REGION Network 65: UNIT 2 STATION 2 MISSING CALIBRATION IN FIXTURE 1 ALARM
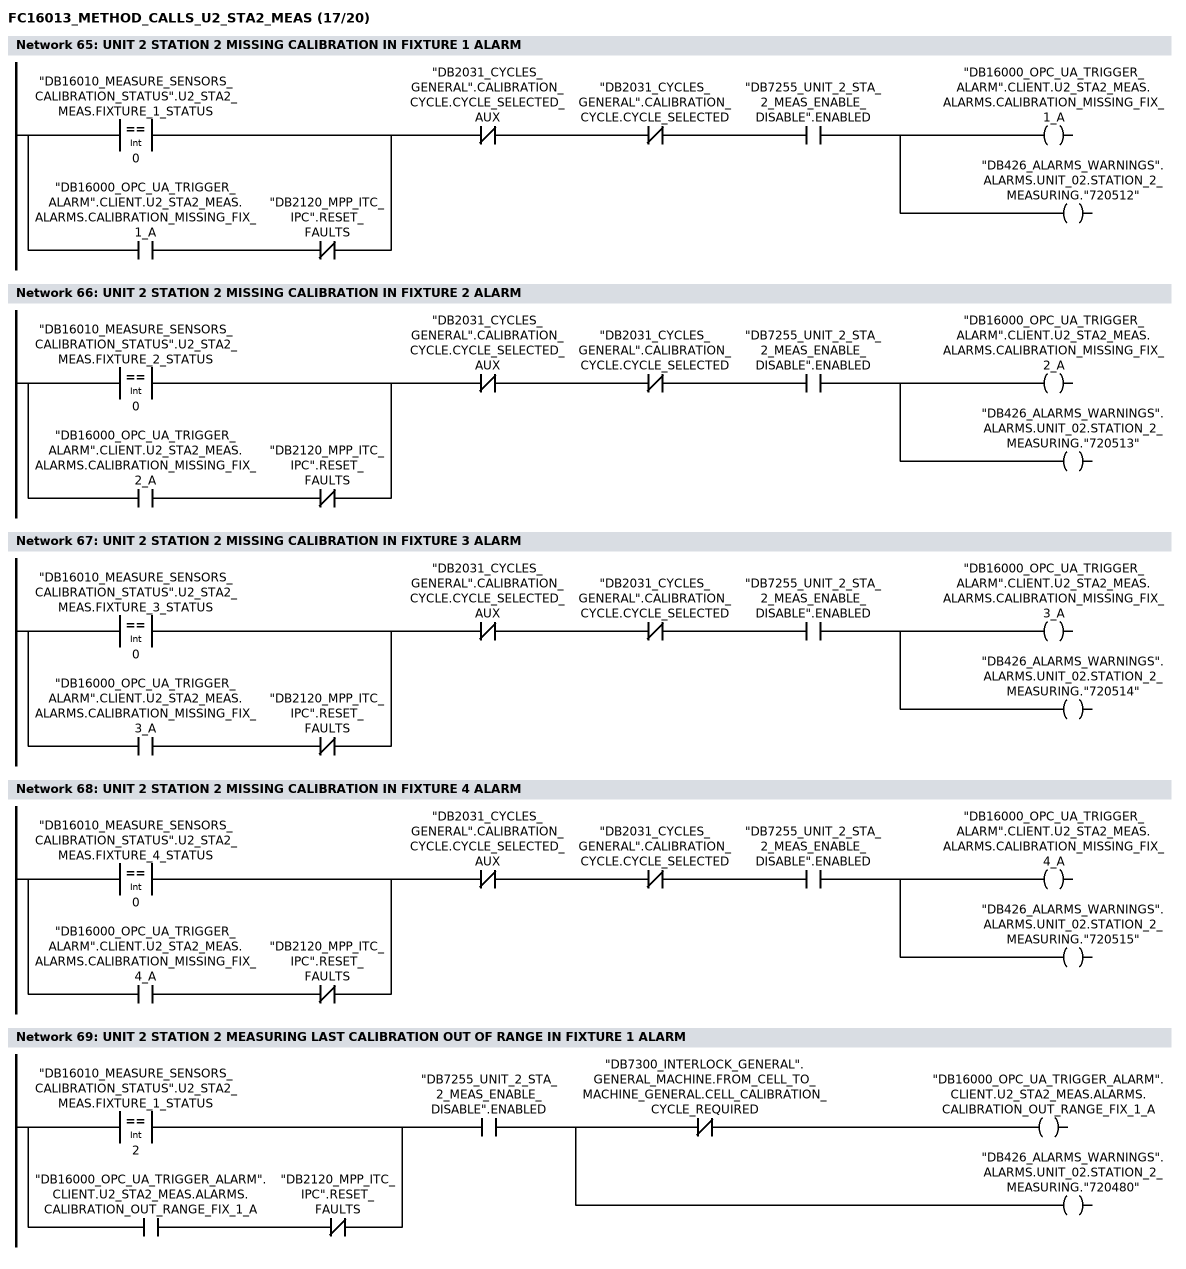
   RUNG wire#powerrail
      { S7_Templates := "SrcType := Int" } EQ_Contact(in1 := "DB16010_MEASURE_SENSORS_CALIBRATION_STATUS".U2_STA2_MEAS.FIXTURE_1_STATUS, in2 := 0)
      wire#w1
      I_Contact( "DB2031_CYCLES_GENERAL".CALIBRATION_CYCLE.CYCLE_SELECTED_AUX )
      I_Contact( "DB2031_CYCLES_GENERAL".CALIBRATION_CYCLE.CYCLE_SELECTED )
      Contact( "DB7255_UNIT_2_STA_2_MEAS_ENABLE_DISABLE".ENABLED )
      wire#w2
      Coil( "DB16000_OPC_UA_TRIGGER_ALARM".CLIENT.U2_STA2_MEAS.ALARMS.CALIBRATION_MISSING_FIX_1_A )
   END_RUNG
   RUNG wire#powerrail
      Contact( "DB16000_OPC_UA_TRIGGER_ALARM".CLIENT.U2_STA2_MEAS.ALARMS.CALIBRATION_MISSING_FIX_1_A )
      I_Contact( "DB2120_MPP_ITC_IPC".RESET_FAULTS )
   END_RUNG wire#w1
   RUNG wire#w2
      Coil( "DB426_ALARMS_WARNINGS".ALARMS.UNIT_02.STATION_2_MEASURING."720512" )
   END_RUNG
   // the same network as SCL:
   "DB16000_OPC_UA_TRIGGER_ALARM".CLIENT.U2_STA2_MEAS.ALARMS.CALIBRATION_MISSING_FIX_1_A := (("DB16010_MEASURE_SENSORS_CALIBRATION_STATUS".U2_STA2_MEAS.FIXTURE_1_STATUS = 0) OR ("DB16000_OPC_UA_TRIGGER_ALARM".CLIENT.U2_STA2_MEAS.ALARMS.CALIBRATION_MISSING_FIX_1_A AND NOT "DB2120_MPP_ITC_IPC".RESET_FAULTS)) AND NOT "DB2031_CYCLES_GENERAL".CALIBRATION_CYCLE.CYCLE_SELECTED_AUX AND NOT "DB2031_CYCLES_GENERAL".CALIBRATION_CYCLE.CYCLE_SELECTED AND "DB7255_UNIT_2_STA_2_MEAS_ENABLE_DISABLE".ENABLED;
   "DB426_ALARMS_WARNINGS".ALARMS.UNIT_02.STATION_2_MEASURING."720512" := "DB16000_OPC_UA_TRIGGER_ALARM".CLIENT.U2_STA2_MEAS.ALARMS.CALIBRATION_MISSING_FIX_1_A;
END_REGION

REGION Network 66: UNIT 2 STATION 2 MISSING CALIBRATION IN FIXTURE 2 ALARM
   RUNG wire#powerrail
      { S7_Templates := "SrcType := Int" } EQ_Contact(in1 := "DB16010_MEASURE_SENSORS_CALIBRATION_STATUS".U2_STA2_MEAS.FIXTURE_2_STATUS, in2 := 0)
      wire#w1
      I_Contact( "DB2031_CYCLES_GENERAL".CALIBRATION_CYCLE.CYCLE_SELECTED_AUX )
      I_Contact( "DB2031_CYCLES_GENERAL".CALIBRATION_CYCLE.CYCLE_SELECTED )
      Contact( "DB7255_UNIT_2_STA_2_MEAS_ENABLE_DISABLE".ENABLED )
      wire#w2
      Coil( "DB16000_OPC_UA_TRIGGER_ALARM".CLIENT.U2_STA2_MEAS.ALARMS.CALIBRATION_MISSING_FIX_2_A )
   END_RUNG
   RUNG wire#powerrail
      Contact( "DB16000_OPC_UA_TRIGGER_ALARM".CLIENT.U2_STA2_MEAS.ALARMS.CALIBRATION_MISSING_FIX_2_A )
      I_Contact( "DB2120_MPP_ITC_IPC".RESET_FAULTS )
   END_RUNG wire#w1
   RUNG wire#w2
      Coil( "DB426_ALARMS_WARNINGS".ALARMS.UNIT_02.STATION_2_MEASURING."720513" )
   END_RUNG
   // the same network as SCL:
   "DB16000_OPC_UA_TRIGGER_ALARM".CLIENT.U2_STA2_MEAS.ALARMS.CALIBRATION_MISSING_FIX_2_A := (("DB16010_MEASURE_SENSORS_CALIBRATION_STATUS".U2_STA2_MEAS.FIXTURE_2_STATUS = 0) OR ("DB16000_OPC_UA_TRIGGER_ALARM".CLIENT.U2_STA2_MEAS.ALARMS.CALIBRATION_MISSING_FIX_2_A AND NOT "DB2120_MPP_ITC_IPC".RESET_FAULTS)) AND NOT "DB2031_CYCLES_GENERAL".CALIBRATION_CYCLE.CYCLE_SELECTED_AUX AND NOT "DB2031_CYCLES_GENERAL".CALIBRATION_CYCLE.CYCLE_SELECTED AND "DB7255_UNIT_2_STA_2_MEAS_ENABLE_DISABLE".ENABLED;
   "DB426_ALARMS_WARNINGS".ALARMS.UNIT_02.STATION_2_MEASURING."720513" := "DB16000_OPC_UA_TRIGGER_ALARM".CLIENT.U2_STA2_MEAS.ALARMS.CALIBRATION_MISSING_FIX_2_A;
END_REGION

REGION Network 67: UNIT 2 STATION 2 MISSING CALIBRATION IN FIXTURE 3 ALARM
   RUNG wire#powerrail
      { S7_Templates := "SrcType := Int" } EQ_Contact(in1 := "DB16010_MEASURE_SENSORS_CALIBRATION_STATUS".U2_STA2_MEAS.FIXTURE_3_STATUS, in2 := 0)
      wire#w1
      I_Contact( "DB2031_CYCLES_GENERAL".CALIBRATION_CYCLE.CYCLE_SELECTED_AUX )
      I_Contact( "DB2031_CYCLES_GENERAL".CALIBRATION_CYCLE.CYCLE_SELECTED )
      Contact( "DB7255_UNIT_2_STA_2_MEAS_ENABLE_DISABLE".ENABLED )
      wire#w2
      Coil( "DB16000_OPC_UA_TRIGGER_ALARM".CLIENT.U2_STA2_MEAS.ALARMS.CALIBRATION_MISSING_FIX_3_A )
   END_RUNG
   RUNG wire#powerrail
      Contact( "DB16000_OPC_UA_TRIGGER_ALARM".CLIENT.U2_STA2_MEAS.ALARMS.CALIBRATION_MISSING_FIX_3_A )
      I_Contact( "DB2120_MPP_ITC_IPC".RESET_FAULTS )
   END_RUNG wire#w1
   RUNG wire#w2
      Coil( "DB426_ALARMS_WARNINGS".ALARMS.UNIT_02.STATION_2_MEASURING."720514" )
   END_RUNG
   // the same network as SCL:
   "DB16000_OPC_UA_TRIGGER_ALARM".CLIENT.U2_STA2_MEAS.ALARMS.CALIBRATION_MISSING_FIX_3_A := (("DB16010_MEASURE_SENSORS_CALIBRATION_STATUS".U2_STA2_MEAS.FIXTURE_3_STATUS = 0) OR ("DB16000_OPC_UA_TRIGGER_ALARM".CLIENT.U2_STA2_MEAS.ALARMS.CALIBRATION_MISSING_FIX_3_A AND NOT "DB2120_MPP_ITC_IPC".RESET_FAULTS)) AND NOT "DB2031_CYCLES_GENERAL".CALIBRATION_CYCLE.CYCLE_SELECTED_AUX AND NOT "DB2031_CYCLES_GENERAL".CALIBRATION_CYCLE.CYCLE_SELECTED AND "DB7255_UNIT_2_STA_2_MEAS_ENABLE_DISABLE".ENABLED;
   "DB426_ALARMS_WARNINGS".ALARMS.UNIT_02.STATION_2_MEASURING."720514" := "DB16000_OPC_UA_TRIGGER_ALARM".CLIENT.U2_STA2_MEAS.ALARMS.CALIBRATION_MISSING_FIX_3_A;
END_REGION

REGION Network 68: UNIT 2 STATION 2 MISSING CALIBRATION IN FIXTURE 4 ALARM
   RUNG wire#powerrail
      { S7_Templates := "SrcType := Int" } EQ_Contact(in1 := "DB16010_MEASURE_SENSORS_CALIBRATION_STATUS".U2_STA2_MEAS.FIXTURE_4_STATUS, in2 := 0)
      wire#w1
      I_Contact( "DB2031_CYCLES_GENERAL".CALIBRATION_CYCLE.CYCLE_SELECTED_AUX )
      I_Contact( "DB2031_CYCLES_GENERAL".CALIBRATION_CYCLE.CYCLE_SELECTED )
      Contact( "DB7255_UNIT_2_STA_2_MEAS_ENABLE_DISABLE".ENABLED )
      wire#w2
      Coil( "DB16000_OPC_UA_TRIGGER_ALARM".CLIENT.U2_STA2_MEAS.ALARMS.CALIBRATION_MISSING_FIX_4_A )
   END_RUNG
   RUNG wire#powerrail
      Contact( "DB16000_OPC_UA_TRIGGER_ALARM".CLIENT.U2_STA2_MEAS.ALARMS.CALIBRATION_MISSING_FIX_4_A )
      I_Contact( "DB2120_MPP_ITC_IPC".RESET_FAULTS )
   END_RUNG wire#w1
   RUNG wire#w2
      Coil( "DB426_ALARMS_WARNINGS".ALARMS.UNIT_02.STATION_2_MEASURING."720515" )
   END_RUNG
   // the same network as SCL:
   "DB16000_OPC_UA_TRIGGER_ALARM".CLIENT.U2_STA2_MEAS.ALARMS.CALIBRATION_MISSING_FIX_4_A := (("DB16010_MEASURE_SENSORS_CALIBRATION_STATUS".U2_STA2_MEAS.FIXTURE_4_STATUS = 0) OR ("DB16000_OPC_UA_TRIGGER_ALARM".CLIENT.U2_STA2_MEAS.ALARMS.CALIBRATION_MISSING_FIX_4_A AND NOT "DB2120_MPP_ITC_IPC".RESET_FAULTS)) AND NOT "DB2031_CYCLES_GENERAL".CALIBRATION_CYCLE.CYCLE_SELECTED_AUX AND NOT "DB2031_CYCLES_GENERAL".CALIBRATION_CYCLE.CYCLE_SELECTED AND "DB7255_UNIT_2_STA_2_MEAS_ENABLE_DISABLE".ENABLED;
   "DB426_ALARMS_WARNINGS".ALARMS.UNIT_02.STATION_2_MEASURING."720515" := "DB16000_OPC_UA_TRIGGER_ALARM".CLIENT.U2_STA2_MEAS.ALARMS.CALIBRATION_MISSING_FIX_4_A;
END_REGION

REGION Network 69: UNIT 2 STATION 2 MEASURING LAST CALIBRATION OUT OF RANGE IN FIXTURE 1 ALARM
   RUNG wire#powerrail
      { S7_Templates := "SrcType := Int" } EQ_Contact(in1 := "DB16010_MEASURE_SENSORS_CALIBRATION_STATUS".U2_STA2_MEAS.FIXTURE_1_STATUS, in2 := 2)
      wire#w1
      Contact( "DB7255_UNIT_2_STA_2_MEAS_ENABLE_DISABLE".ENABLED )
      wire#w2
      I_Contact( "DB7300_INTERLOCK_GENERAL".GENERAL_MACHINE.FROM_CELL_TO_MACHINE_GENERAL.CELL_CALIBRATION_CYCLE_REQUIRED )
      Coil( "DB16000_OPC_UA_TRIGGER_ALARM".CLIENT.U2_STA2_MEAS.ALARMS.CALIBRATION_OUT_RANGE_FIX_1_A )
   END_RUNG
   RUNG wire#powerrail
      Contact( "DB16000_OPC_UA_TRIGGER_ALARM".CLIENT.U2_STA2_MEAS.ALARMS.CALIBRATION_OUT_RANGE_FIX_1_A )
      I_Contact( "DB2120_MPP_ITC_IPC".RESET_FAULTS )
   END_RUNG wire#w1
   RUNG wire#w2
      Coil( "DB426_ALARMS_WARNINGS".ALARMS.UNIT_02.STATION_2_MEASURING."720480" )
   END_RUNG
   // the same network as SCL:
   #_w1 := (("DB16010_MEASURE_SENSORS_CALIBRATION_STATUS".U2_STA2_MEAS.FIXTURE_1_STATUS = 2) OR ("DB16000_OPC_UA_TRIGGER_ALARM".CLIENT.U2_STA2_MEAS.ALARMS.CALIBRATION_OUT_RANGE_FIX_1_A AND NOT "DB2120_MPP_ITC_IPC".RESET_FAULTS)) AND "DB7255_UNIT_2_STA_2_MEAS_ENABLE_DISABLE".ENABLED;
   "DB16000_OPC_UA_TRIGGER_ALARM".CLIENT.U2_STA2_MEAS.ALARMS.CALIBRATION_OUT_RANGE_FIX_1_A := #_w1 AND NOT "DB7300_INTERLOCK_GENERAL".GENERAL_MACHINE.FROM_CELL_TO_MACHINE_GENERAL.CELL_CALIBRATION_CYCLE_REQUIRED;
   "DB426_ALARMS_WARNINGS".ALARMS.UNIT_02.STATION_2_MEASURING."720480" := #_w1;
END_REGION

REGION Network 70: UNIT 2 STATION 2 MEASURING LAST CALIBRATION OUT OF RANGE IN FIXTURE 2 ALARM
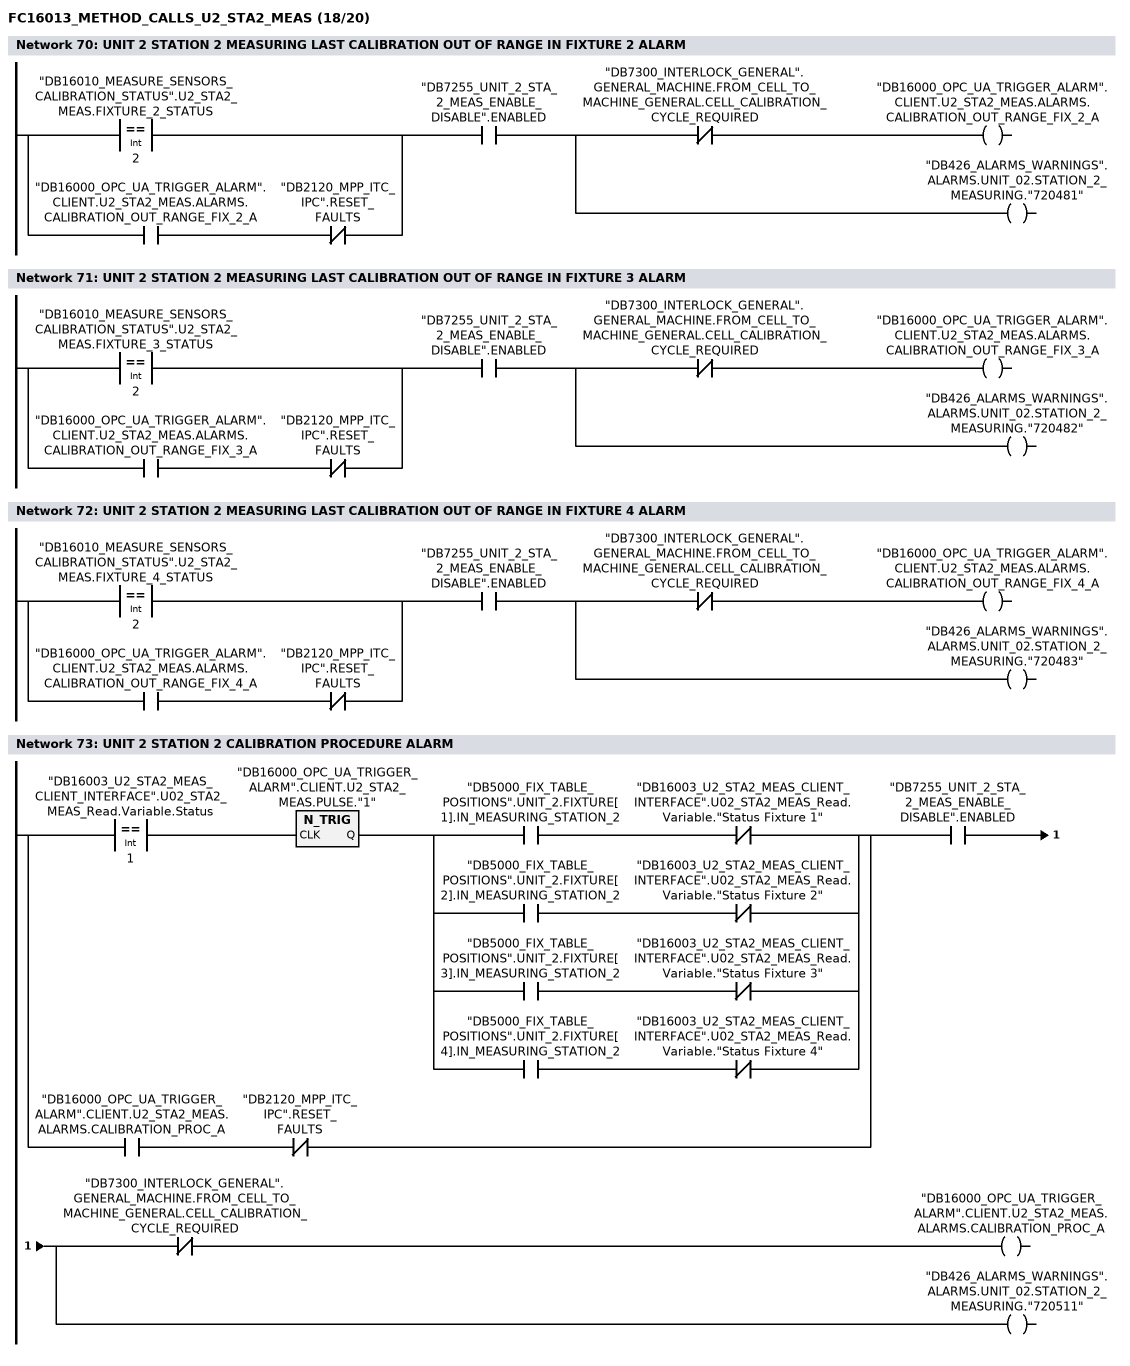
   RUNG wire#powerrail
      { S7_Templates := "SrcType := Int" } EQ_Contact(in1 := "DB16010_MEASURE_SENSORS_CALIBRATION_STATUS".U2_STA2_MEAS.FIXTURE_2_STATUS, in2 := 2)
      wire#w1
      Contact( "DB7255_UNIT_2_STA_2_MEAS_ENABLE_DISABLE".ENABLED )
      wire#w2
      I_Contact( "DB7300_INTERLOCK_GENERAL".GENERAL_MACHINE.FROM_CELL_TO_MACHINE_GENERAL.CELL_CALIBRATION_CYCLE_REQUIRED )
      Coil( "DB16000_OPC_UA_TRIGGER_ALARM".CLIENT.U2_STA2_MEAS.ALARMS.CALIBRATION_OUT_RANGE_FIX_2_A )
   END_RUNG
   RUNG wire#powerrail
      Contact( "DB16000_OPC_UA_TRIGGER_ALARM".CLIENT.U2_STA2_MEAS.ALARMS.CALIBRATION_OUT_RANGE_FIX_2_A )
      I_Contact( "DB2120_MPP_ITC_IPC".RESET_FAULTS )
   END_RUNG wire#w1
   RUNG wire#w2
      Coil( "DB426_ALARMS_WARNINGS".ALARMS.UNIT_02.STATION_2_MEASURING."720481" )
   END_RUNG
   // the same network as SCL:
   #_w1 := (("DB16010_MEASURE_SENSORS_CALIBRATION_STATUS".U2_STA2_MEAS.FIXTURE_2_STATUS = 2) OR ("DB16000_OPC_UA_TRIGGER_ALARM".CLIENT.U2_STA2_MEAS.ALARMS.CALIBRATION_OUT_RANGE_FIX_2_A AND NOT "DB2120_MPP_ITC_IPC".RESET_FAULTS)) AND "DB7255_UNIT_2_STA_2_MEAS_ENABLE_DISABLE".ENABLED;
   "DB16000_OPC_UA_TRIGGER_ALARM".CLIENT.U2_STA2_MEAS.ALARMS.CALIBRATION_OUT_RANGE_FIX_2_A := #_w1 AND NOT "DB7300_INTERLOCK_GENERAL".GENERAL_MACHINE.FROM_CELL_TO_MACHINE_GENERAL.CELL_CALIBRATION_CYCLE_REQUIRED;
   "DB426_ALARMS_WARNINGS".ALARMS.UNIT_02.STATION_2_MEASURING."720481" := #_w1;
END_REGION

REGION Network 71: UNIT 2 STATION 2 MEASURING LAST CALIBRATION OUT OF RANGE IN FIXTURE 3 ALARM
   RUNG wire#powerrail
      { S7_Templates := "SrcType := Int" } EQ_Contact(in1 := "DB16010_MEASURE_SENSORS_CALIBRATION_STATUS".U2_STA2_MEAS.FIXTURE_3_STATUS, in2 := 2)
      wire#w1
      Contact( "DB7255_UNIT_2_STA_2_MEAS_ENABLE_DISABLE".ENABLED )
      wire#w2
      I_Contact( "DB7300_INTERLOCK_GENERAL".GENERAL_MACHINE.FROM_CELL_TO_MACHINE_GENERAL.CELL_CALIBRATION_CYCLE_REQUIRED )
      Coil( "DB16000_OPC_UA_TRIGGER_ALARM".CLIENT.U2_STA2_MEAS.ALARMS.CALIBRATION_OUT_RANGE_FIX_3_A )
   END_RUNG
   RUNG wire#powerrail
      Contact( "DB16000_OPC_UA_TRIGGER_ALARM".CLIENT.U2_STA2_MEAS.ALARMS.CALIBRATION_OUT_RANGE_FIX_3_A )
      I_Contact( "DB2120_MPP_ITC_IPC".RESET_FAULTS )
   END_RUNG wire#w1
   RUNG wire#w2
      Coil( "DB426_ALARMS_WARNINGS".ALARMS.UNIT_02.STATION_2_MEASURING."720482" )
   END_RUNG
   // the same network as SCL:
   #_w1 := (("DB16010_MEASURE_SENSORS_CALIBRATION_STATUS".U2_STA2_MEAS.FIXTURE_3_STATUS = 2) OR ("DB16000_OPC_UA_TRIGGER_ALARM".CLIENT.U2_STA2_MEAS.ALARMS.CALIBRATION_OUT_RANGE_FIX_3_A AND NOT "DB2120_MPP_ITC_IPC".RESET_FAULTS)) AND "DB7255_UNIT_2_STA_2_MEAS_ENABLE_DISABLE".ENABLED;
   "DB16000_OPC_UA_TRIGGER_ALARM".CLIENT.U2_STA2_MEAS.ALARMS.CALIBRATION_OUT_RANGE_FIX_3_A := #_w1 AND NOT "DB7300_INTERLOCK_GENERAL".GENERAL_MACHINE.FROM_CELL_TO_MACHINE_GENERAL.CELL_CALIBRATION_CYCLE_REQUIRED;
   "DB426_ALARMS_WARNINGS".ALARMS.UNIT_02.STATION_2_MEASURING."720482" := #_w1;
END_REGION

REGION Network 72: UNIT 2 STATION 2 MEASURING LAST CALIBRATION OUT OF RANGE IN FIXTURE 4 ALARM
   RUNG wire#powerrail
      { S7_Templates := "SrcType := Int" } EQ_Contact(in1 := "DB16010_MEASURE_SENSORS_CALIBRATION_STATUS".U2_STA2_MEAS.FIXTURE_4_STATUS, in2 := 2)
      wire#w1
      Contact( "DB7255_UNIT_2_STA_2_MEAS_ENABLE_DISABLE".ENABLED )
      wire#w2
      I_Contact( "DB7300_INTERLOCK_GENERAL".GENERAL_MACHINE.FROM_CELL_TO_MACHINE_GENERAL.CELL_CALIBRATION_CYCLE_REQUIRED )
      Coil( "DB16000_OPC_UA_TRIGGER_ALARM".CLIENT.U2_STA2_MEAS.ALARMS.CALIBRATION_OUT_RANGE_FIX_4_A )
   END_RUNG
   RUNG wire#powerrail
      Contact( "DB16000_OPC_UA_TRIGGER_ALARM".CLIENT.U2_STA2_MEAS.ALARMS.CALIBRATION_OUT_RANGE_FIX_4_A )
      I_Contact( "DB2120_MPP_ITC_IPC".RESET_FAULTS )
   END_RUNG wire#w1
   RUNG wire#w2
      Coil( "DB426_ALARMS_WARNINGS".ALARMS.UNIT_02.STATION_2_MEASURING."720483" )
   END_RUNG
   // the same network as SCL:
   #_w1 := (("DB16010_MEASURE_SENSORS_CALIBRATION_STATUS".U2_STA2_MEAS.FIXTURE_4_STATUS = 2) OR ("DB16000_OPC_UA_TRIGGER_ALARM".CLIENT.U2_STA2_MEAS.ALARMS.CALIBRATION_OUT_RANGE_FIX_4_A AND NOT "DB2120_MPP_ITC_IPC".RESET_FAULTS)) AND "DB7255_UNIT_2_STA_2_MEAS_ENABLE_DISABLE".ENABLED;
   "DB16000_OPC_UA_TRIGGER_ALARM".CLIENT.U2_STA2_MEAS.ALARMS.CALIBRATION_OUT_RANGE_FIX_4_A := #_w1 AND NOT "DB7300_INTERLOCK_GENERAL".GENERAL_MACHINE.FROM_CELL_TO_MACHINE_GENERAL.CELL_CALIBRATION_CYCLE_REQUIRED;
   "DB426_ALARMS_WARNINGS".ALARMS.UNIT_02.STATION_2_MEASURING."720483" := #_w1;
END_REGION

REGION Network 73: UNIT 2 STATION 2 CALIBRATION PROCEDURE ALARM
   RUNG wire#powerrail
      { S7_Templates := "SrcType := Int" } EQ_Contact(in1 := "DB16003_U2_STA2_MEAS_CLIENT_INTERFACE".U02_STA2_MEAS_Read.Variable.Status, in2 := 1)
      N_Trig( "DB16000_OPC_UA_TRIGGER_ALARM".CLIENT.U2_STA2_MEAS.PULSE."1" )
      wire#w1
      Contact( "DB5000_FIX_TABLE_POSITIONS".UNIT_2.FIXTURE[1].IN_MEASURING_STATION_2 )
      I_Contact( "DB16003_U2_STA2_MEAS_CLIENT_INTERFACE".U02_STA2_MEAS_Read.Variable."Status Fixture 1" )
      wire#w2
      Contact( "DB7255_UNIT_2_STA_2_MEAS_ENABLE_DISABLE".ENABLED )
      wire#w3
      I_Contact( "DB7300_INTERLOCK_GENERAL".GENERAL_MACHINE.FROM_CELL_TO_MACHINE_GENERAL.CELL_CALIBRATION_CYCLE_REQUIRED )
      Coil( "DB16000_OPC_UA_TRIGGER_ALARM".CLIENT.U2_STA2_MEAS.ALARMS.CALIBRATION_PROC_A )
   END_RUNG
   RUNG wire#w1
      Contact( "DB5000_FIX_TABLE_POSITIONS".UNIT_2.FIXTURE[2].IN_MEASURING_STATION_2 )
      I_Contact( "DB16003_U2_STA2_MEAS_CLIENT_INTERFACE".U02_STA2_MEAS_Read.Variable."Status Fixture 2" )
   END_RUNG wire#w2
   RUNG wire#w1
      Contact( "DB5000_FIX_TABLE_POSITIONS".UNIT_2.FIXTURE[3].IN_MEASURING_STATION_2 )
      I_Contact( "DB16003_U2_STA2_MEAS_CLIENT_INTERFACE".U02_STA2_MEAS_Read.Variable."Status Fixture 3" )
   END_RUNG wire#w2
   RUNG wire#w1
      Contact( "DB5000_FIX_TABLE_POSITIONS".UNIT_2.FIXTURE[4].IN_MEASURING_STATION_2 )
      I_Contact( "DB16003_U2_STA2_MEAS_CLIENT_INTERFACE".U02_STA2_MEAS_Read.Variable."Status Fixture 4" )
   END_RUNG wire#w2
   RUNG wire#powerrail
      Contact( "DB16000_OPC_UA_TRIGGER_ALARM".CLIENT.U2_STA2_MEAS.ALARMS.CALIBRATION_PROC_A )
      I_Contact( "DB2120_MPP_ITC_IPC".RESET_FAULTS )
   END_RUNG wire#w2
   RUNG wire#w3
      Coil( "DB426_ALARMS_WARNINGS".ALARMS.UNIT_02.STATION_2_MEASURING."720511" )
   END_RUNG
   // the same network as SCL:
   #_w1 := "DB16003_U2_STA2_MEAS_CLIENT_INTERFACE".U02_STA2_MEAS_Read.Variable.Status = 1;
   #_w2 := NOT #_w1 AND "DB16000_OPC_UA_TRIGGER_ALARM".CLIENT.U2_STA2_MEAS.PULSE."1";   // falling edge
   "DB16000_OPC_UA_TRIGGER_ALARM".CLIENT.U2_STA2_MEAS.PULSE."1" := #_w1;
   #_w3 := ((#_w2 AND (("DB5000_FIX_TABLE_POSITIONS".UNIT_2.FIXTURE[1].IN_MEASURING_STATION_2 AND NOT "DB16003_U2_STA2_MEAS_CLIENT_INTERFACE".U02_STA2_MEAS_Read.Variable."Status Fixture 1") OR ("DB5000_FIX_TABLE_POSITIONS".UNIT_2.FIXTURE[2].IN_MEASURING_STATION_2 AND NOT "DB16003_U2_STA2_MEAS_CLIENT_INTERFACE".U02_STA2_MEAS_Read.Variable."Status Fixture 2") OR ("DB5000_FIX_TABLE_POSITIONS".UNIT_2.FIXTURE[3].IN_MEASURING_STATION_2 AND NOT "DB16003_U2_STA2_MEAS_CLIENT_INTERFACE".U02_STA2_MEAS_Read.Variable."Status Fixture 3") OR ("DB5000_FIX_TABLE_POSITIONS".UNIT_2.FIXTURE[4].IN_MEASURING_STATION_2 AND NOT "DB16003_U2_STA2_MEAS_CLIENT_INTERFACE".U02_STA2_MEAS_Read.Variable."Status Fixture 4"))) OR ("DB16000_OPC_UA_TRIGGER_ALARM".CLIENT.U2_STA2_MEAS.ALARMS.CALIBRATION_PROC_A AND NOT "DB2120_MPP_ITC_IPC".RESET_FAULTS)) AND "DB7255_UNIT_2_STA_2_MEAS_ENABLE_DISABLE".ENABLED;
   "DB16000_OPC_UA_TRIGGER_ALARM".CLIENT.U2_STA2_MEAS.ALARMS.CALIBRATION_PROC_A := #_w3 AND NOT "DB7300_INTERLOCK_GENERAL".GENERAL_MACHINE.FROM_CELL_TO_MACHINE_GENERAL.CELL_CALIBRATION_CYCLE_REQUIRED;
   "DB426_ALARMS_WARNINGS".ALARMS.UNIT_02.STATION_2_MEASURING."720511" := #_w3;
END_REGION

REGION Network 74: UNIT 2 STATION 2 MEASURING INITIALIZING SENSOR ALARM
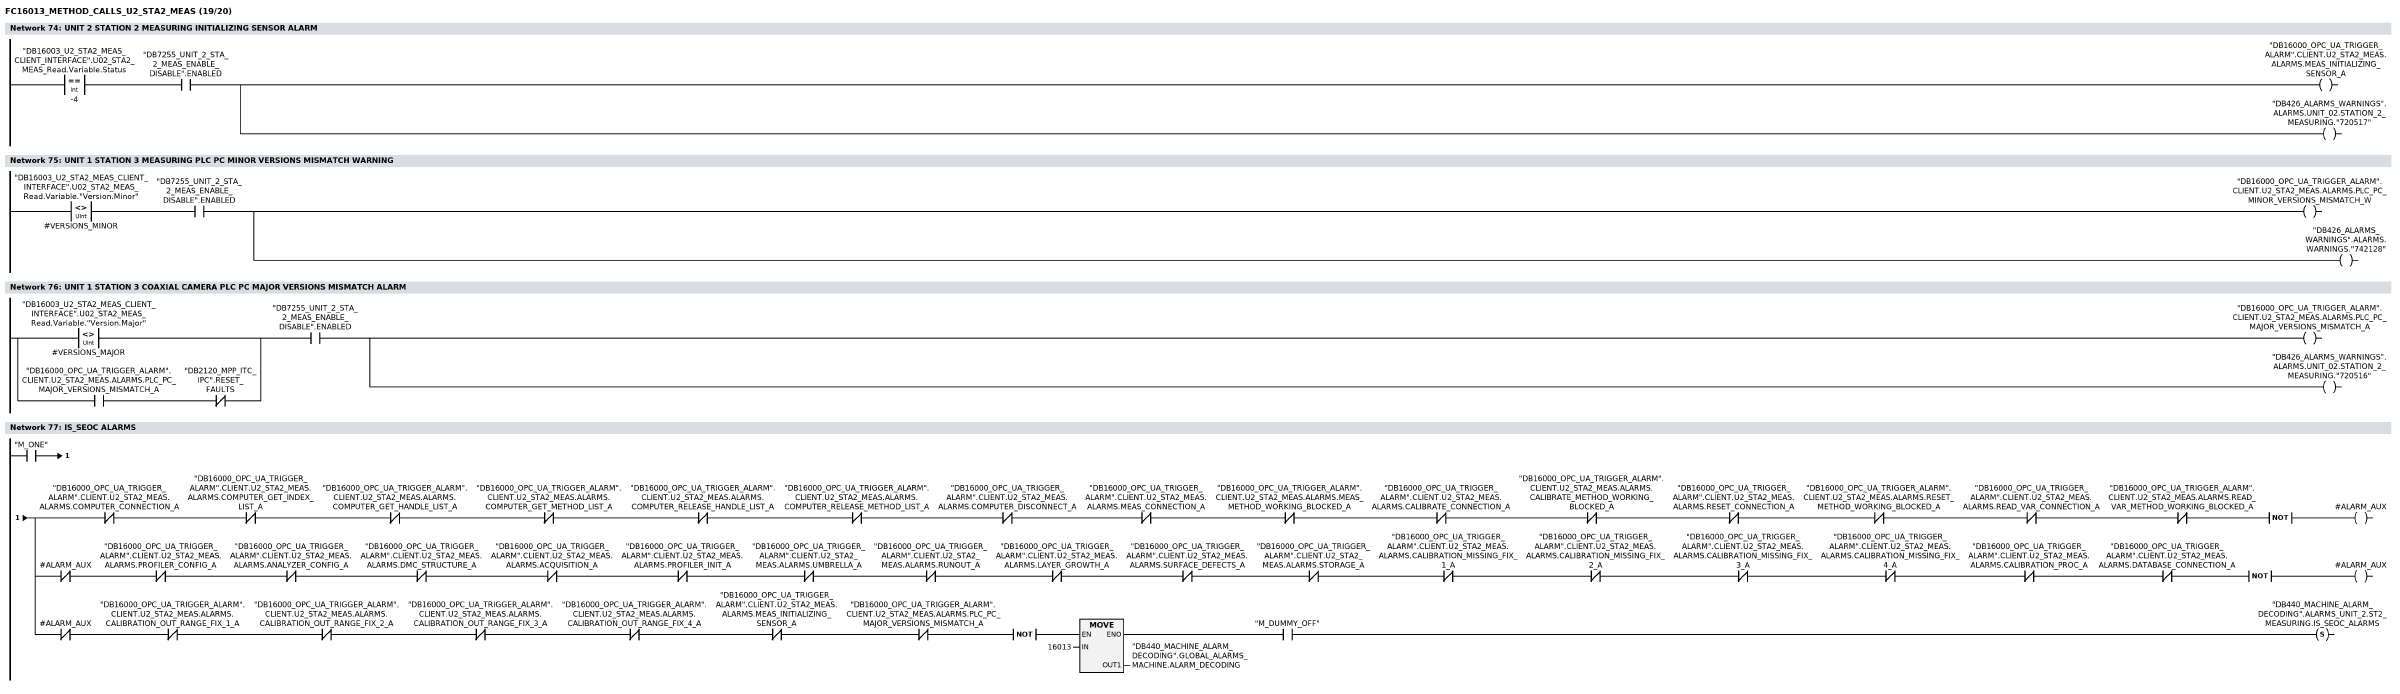
   RUNG wire#powerrail
      { S7_Templates := "SrcType := Int" } EQ_Contact(in1 := "DB16003_U2_STA2_MEAS_CLIENT_INTERFACE".U02_STA2_MEAS_Read.Variable.Status, in2 := -4)
      Contact( "DB7255_UNIT_2_STA_2_MEAS_ENABLE_DISABLE".ENABLED )
      wire#w1
      Coil( "DB16000_OPC_UA_TRIGGER_ALARM".CLIENT.U2_STA2_MEAS.ALARMS.MEAS_INITIALIZING_SENSOR_A )
   END_RUNG
   RUNG wire#w1
      Coil( "DB426_ALARMS_WARNINGS".ALARMS.UNIT_02.STATION_2_MEASURING."720517" )
   END_RUNG
   // the same network as SCL:
   "DB16000_OPC_UA_TRIGGER_ALARM".CLIENT.U2_STA2_MEAS.ALARMS.MEAS_INITIALIZING_SENSOR_A := ("DB16003_U2_STA2_MEAS_CLIENT_INTERFACE".U02_STA2_MEAS_Read.Variable.Status = (-4)) AND "DB7255_UNIT_2_STA_2_MEAS_ENABLE_DISABLE".ENABLED;
   "DB426_ALARMS_WARNINGS".ALARMS.UNIT_02.STATION_2_MEASURING."720517" := "DB16000_OPC_UA_TRIGGER_ALARM".CLIENT.U2_STA2_MEAS.ALARMS.MEAS_INITIALIZING_SENSOR_A;
END_REGION

REGION Network 75: UNIT 1 STATION 3 MEASURING PLC PC MINOR VERSIONS MISMATCH WARNING
   RUNG wire#powerrail
      { S7_Templates := "SrcType := UInt" } NE_Contact(in1 := "DB16003_U2_STA2_MEAS_CLIENT_INTERFACE".U02_STA2_MEAS_Read.Variable."Version.Minor", in2 := #VERSIONS_MINOR)
      Contact( "DB7255_UNIT_2_STA_2_MEAS_ENABLE_DISABLE".ENABLED )
      wire#w1
      Coil( "DB16000_OPC_UA_TRIGGER_ALARM".CLIENT.U2_STA2_MEAS.ALARMS.PLC_PC_MINOR_VERSIONS_MISMATCH_W )
   END_RUNG
   RUNG wire#w1
      Coil( "DB426_ALARMS_WARNINGS".ALARMS.WARNINGS."742128" )
   END_RUNG
   // the same network as SCL:
   "DB16000_OPC_UA_TRIGGER_ALARM".CLIENT.U2_STA2_MEAS.ALARMS.PLC_PC_MINOR_VERSIONS_MISMATCH_W := ("DB16003_U2_STA2_MEAS_CLIENT_INTERFACE".U02_STA2_MEAS_Read.Variable."Version.Minor" <> #VERSIONS_MINOR) AND "DB7255_UNIT_2_STA_2_MEAS_ENABLE_DISABLE".ENABLED;
   "DB426_ALARMS_WARNINGS".ALARMS.WARNINGS."742128" := "DB16000_OPC_UA_TRIGGER_ALARM".CLIENT.U2_STA2_MEAS.ALARMS.PLC_PC_MINOR_VERSIONS_MISMATCH_W;
END_REGION

REGION Network 76: UNIT 1 STATION 3 COAXIAL CAMERA PLC PC MAJOR VERSIONS MISMATCH ALARM
   RUNG wire#powerrail
      { S7_Templates := "SrcType := UInt" } NE_Contact(in1 := "DB16003_U2_STA2_MEAS_CLIENT_INTERFACE".U02_STA2_MEAS_Read.Variable."Version.Major", in2 := #VERSIONS_MAJOR)
      wire#w1
      Contact( "DB7255_UNIT_2_STA_2_MEAS_ENABLE_DISABLE".ENABLED )
      wire#w2
      Coil( "DB16000_OPC_UA_TRIGGER_ALARM".CLIENT.U2_STA2_MEAS.ALARMS.PLC_PC_MAJOR_VERSIONS_MISMATCH_A )
   END_RUNG
   RUNG wire#powerrail
      Contact( "DB16000_OPC_UA_TRIGGER_ALARM".CLIENT.U2_STA2_MEAS.ALARMS.PLC_PC_MAJOR_VERSIONS_MISMATCH_A )
      I_Contact( "DB2120_MPP_ITC_IPC".RESET_FAULTS )
   END_RUNG wire#w1
   RUNG wire#w2
      Coil( "DB426_ALARMS_WARNINGS".ALARMS.UNIT_02.STATION_2_MEASURING."720516" )
   END_RUNG
   // the same network as SCL:
   "DB16000_OPC_UA_TRIGGER_ALARM".CLIENT.U2_STA2_MEAS.ALARMS.PLC_PC_MAJOR_VERSIONS_MISMATCH_A := (("DB16003_U2_STA2_MEAS_CLIENT_INTERFACE".U02_STA2_MEAS_Read.Variable."Version.Major" <> #VERSIONS_MAJOR) OR ("DB16000_OPC_UA_TRIGGER_ALARM".CLIENT.U2_STA2_MEAS.ALARMS.PLC_PC_MAJOR_VERSIONS_MISMATCH_A AND NOT "DB2120_MPP_ITC_IPC".RESET_FAULTS)) AND "DB7255_UNIT_2_STA_2_MEAS_ENABLE_DISABLE".ENABLED;
   "DB426_ALARMS_WARNINGS".ALARMS.UNIT_02.STATION_2_MEASURING."720516" := "DB16000_OPC_UA_TRIGGER_ALARM".CLIENT.U2_STA2_MEAS.ALARMS.PLC_PC_MAJOR_VERSIONS_MISMATCH_A;
END_REGION

REGION Network 77: IS_SEOC ALARMS
   RUNG wire#powerrail
      Contact( "M_ONE" )
      wire#w1
      I_Contact( "DB16000_OPC_UA_TRIGGER_ALARM".CLIENT.U2_STA2_MEAS.ALARMS.COMPUTER_CONNECTION_A )
      I_Contact( "DB16000_OPC_UA_TRIGGER_ALARM".CLIENT.U2_STA2_MEAS.ALARMS.COMPUTER_GET_INDEX_LIST_A )
      I_Contact( "DB16000_OPC_UA_TRIGGER_ALARM".CLIENT.U2_STA2_MEAS.ALARMS.COMPUTER_GET_HANDLE_LIST_A )
      I_Contact( "DB16000_OPC_UA_TRIGGER_ALARM".CLIENT.U2_STA2_MEAS.ALARMS.COMPUTER_GET_METHOD_LIST_A )
      I_Contact( "DB16000_OPC_UA_TRIGGER_ALARM".CLIENT.U2_STA2_MEAS.ALARMS.COMPUTER_RELEASE_HANDLE_LIST_A )
      I_Contact( "DB16000_OPC_UA_TRIGGER_ALARM".CLIENT.U2_STA2_MEAS.ALARMS.COMPUTER_RELEASE_METHOD_LIST_A )
      I_Contact( "DB16000_OPC_UA_TRIGGER_ALARM".CLIENT.U2_STA2_MEAS.ALARMS.COMPUTER_DISCONNECT_A )
      I_Contact( "DB16000_OPC_UA_TRIGGER_ALARM".CLIENT.U2_STA2_MEAS.ALARMS.MEAS_CONNECTION_A )
      I_Contact( "DB16000_OPC_UA_TRIGGER_ALARM".CLIENT.U2_STA2_MEAS.ALARMS.MEAS_METHOD_WORKING_BLOCKED_A )
      I_Contact( "DB16000_OPC_UA_TRIGGER_ALARM".CLIENT.U2_STA2_MEAS.ALARMS.CALIBRATE_CONNECTION_A )
      I_Contact( "DB16000_OPC_UA_TRIGGER_ALARM".CLIENT.U2_STA2_MEAS.ALARMS.CALIBRATE_METHOD_WORKING_BLOCKED_A )
      I_Contact( "DB16000_OPC_UA_TRIGGER_ALARM".CLIENT.U2_STA2_MEAS.ALARMS.RESET_CONNECTION_A )
      I_Contact( "DB16000_OPC_UA_TRIGGER_ALARM".CLIENT.U2_STA2_MEAS.ALARMS.RESET_METHOD_WORKING_BLOCKED_A )
      I_Contact( "DB16000_OPC_UA_TRIGGER_ALARM".CLIENT.U2_STA2_MEAS.ALARMS.READ_VAR_CONNECTION_A )
      I_Contact( "DB16000_OPC_UA_TRIGGER_ALARM".CLIENT.U2_STA2_MEAS.ALARMS.READ_VAR_METHOD_WORKING_BLOCKED_A )
      Not()
      Coil( #ALARM_AUX )
   END_RUNG
   RUNG wire#w1
      I_Contact( #ALARM_AUX )
      I_Contact( "DB16000_OPC_UA_TRIGGER_ALARM".CLIENT.U2_STA2_MEAS.ALARMS.PROFILER_CONFIG_A )
      I_Contact( "DB16000_OPC_UA_TRIGGER_ALARM".CLIENT.U2_STA2_MEAS.ALARMS.ANALYZER_CONFIG_A )
      I_Contact( "DB16000_OPC_UA_TRIGGER_ALARM".CLIENT.U2_STA2_MEAS.ALARMS.DMC_STRUCTURE_A )
      I_Contact( "DB16000_OPC_UA_TRIGGER_ALARM".CLIENT.U2_STA2_MEAS.ALARMS.ACQUISITION_A )
      I_Contact( "DB16000_OPC_UA_TRIGGER_ALARM".CLIENT.U2_STA2_MEAS.ALARMS.PROFILER_INIT_A )
      I_Contact( "DB16000_OPC_UA_TRIGGER_ALARM".CLIENT.U2_STA2_MEAS.ALARMS.UMBRELLA_A )
      I_Contact( "DB16000_OPC_UA_TRIGGER_ALARM".CLIENT.U2_STA2_MEAS.ALARMS.RUNOUT_A )
      I_Contact( "DB16000_OPC_UA_TRIGGER_ALARM".CLIENT.U2_STA2_MEAS.ALARMS.LAYER_GROWTH_A )
      I_Contact( "DB16000_OPC_UA_TRIGGER_ALARM".CLIENT.U2_STA2_MEAS.ALARMS.SURFACE_DEFECTS_A )
      I_Contact( "DB16000_OPC_UA_TRIGGER_ALARM".CLIENT.U2_STA2_MEAS.ALARMS.STORAGE_A )
      I_Contact( "DB16000_OPC_UA_TRIGGER_ALARM".CLIENT.U2_STA2_MEAS.ALARMS.CALIBRATION_MISSING_FIX_1_A )
      I_Contact( "DB16000_OPC_UA_TRIGGER_ALARM".CLIENT.U2_STA2_MEAS.ALARMS.CALIBRATION_MISSING_FIX_2_A )
      I_Contact( "DB16000_OPC_UA_TRIGGER_ALARM".CLIENT.U2_STA2_MEAS.ALARMS.CALIBRATION_MISSING_FIX_3_A )
      I_Contact( "DB16000_OPC_UA_TRIGGER_ALARM".CLIENT.U2_STA2_MEAS.ALARMS.CALIBRATION_MISSING_FIX_4_A )
      I_Contact( "DB16000_OPC_UA_TRIGGER_ALARM".CLIENT.U2_STA2_MEAS.ALARMS.CALIBRATION_PROC_A )
      I_Contact( "DB16000_OPC_UA_TRIGGER_ALARM".CLIENT.U2_STA2_MEAS.ALARMS.DATABASE_CONNECTION_A )
      Not()
      Coil( #ALARM_AUX )
   END_RUNG
   RUNG wire#w1
      I_Contact( #ALARM_AUX )
      I_Contact( "DB16000_OPC_UA_TRIGGER_ALARM".CLIENT.U2_STA2_MEAS.ALARMS.CALIBRATION_OUT_RANGE_FIX_1_A )
      I_Contact( "DB16000_OPC_UA_TRIGGER_ALARM".CLIENT.U2_STA2_MEAS.ALARMS.CALIBRATION_OUT_RANGE_FIX_2_A )
      I_Contact( "DB16000_OPC_UA_TRIGGER_ALARM".CLIENT.U2_STA2_MEAS.ALARMS.CALIBRATION_OUT_RANGE_FIX_3_A )
      I_Contact( "DB16000_OPC_UA_TRIGGER_ALARM".CLIENT.U2_STA2_MEAS.ALARMS.CALIBRATION_OUT_RANGE_FIX_4_A )
      I_Contact( "DB16000_OPC_UA_TRIGGER_ALARM".CLIENT.U2_STA2_MEAS.ALARMS.MEAS_INITIALIZING_SENSOR_A )
      I_Contact( "DB16000_OPC_UA_TRIGGER_ALARM".CLIENT.U2_STA2_MEAS.ALARMS.PLC_PC_MAJOR_VERSIONS_MISMATCH_A )
      Not()
      Move(in := 16013, out1 => "DB440_MACHINE_ALARM_DECODING".GLOBAL_ALARMS_MACHINE.ALARM_DECODING)
      Contact( "M_DUMMY_OFF" )
      S_Coil( "DB440_MACHINE_ALARM_DECODING".ALARMS_UNIT_2.ST2_MEASURING.IS_SEOC_ALARMS )
   END_RUNG
   // the same network as SCL:
   #ALARM_AUX := NOT ("M_ONE" AND NOT "DB16000_OPC_UA_TRIGGER_ALARM".CLIENT.U2_STA2_MEAS.ALARMS.COMPUTER_CONNECTION_A AND NOT "DB16000_OPC_UA_TRIGGER_ALARM".CLIENT.U2_STA2_MEAS.ALARMS.COMPUTER_GET_INDEX_LIST_A AND NOT "DB16000_OPC_UA_TRIGGER_ALARM".CLIENT.U2_STA2_MEAS.ALARMS.COMPUTER_GET_HANDLE_LIST_A AND NOT "DB16000_OPC_UA_TRIGGER_ALARM".CLIENT.U2_STA2_MEAS.ALARMS.COMPUTER_GET_METHOD_LIST_A AND NOT "DB16000_OPC_UA_TRIGGER_ALARM".CLIENT.U2_STA2_MEAS.ALARMS.COMPUTER_RELEASE_HANDLE_LIST_A AND NOT "DB16000_OPC_UA_TRIGGER_ALARM".CLIENT.U2_STA2_MEAS.ALARMS.COMPUTER_RELEASE_METHOD_LIST_A AND NOT "DB16000_OPC_UA_TRIGGER_ALARM".CLIENT.U2_STA2_MEAS.ALARMS.COMPUTER_DISCONNECT_A AND NOT "DB16000_OPC_UA_TRIGGER_ALARM".CLIENT.U2_STA2_MEAS.ALARMS.MEAS_CONNECTION_A AND NOT "DB16000_OPC_UA_TRIGGER_ALARM".CLIENT.U2_STA2_MEAS.ALARMS.MEAS_METHOD_WORKING_BLOCKED_A AND NOT "DB16000_OPC_UA_TRIGGER_ALARM".CLIENT.U2_STA2_MEAS.ALARMS.CALIBRATE_CONNECTION_A AND NOT "DB16000_OPC_UA_TRIGGER_ALARM".CLIENT.U2_STA2_MEAS.ALARMS.CALIBRATE_METHOD_WORKING_BLOCKED_A AND NOT "DB16000_OPC_UA_TRIGGER_ALARM".CLIENT.U2_STA2_MEAS.ALARMS.RESET_CONNECTION_A AND NOT "DB16000_OPC_UA_TRIGGER_ALARM".CLIENT.U2_STA2_MEAS.ALARMS.RESET_METHOD_WORKING_BLOCKED_A AND NOT "DB16000_OPC_UA_TRIGGER_ALARM".CLIENT.U2_STA2_MEAS.ALARMS.READ_VAR_CONNECTION_A AND NOT "DB16000_OPC_UA_TRIGGER_ALARM".CLIENT.U2_STA2_MEAS.ALARMS.READ_VAR_METHOD_WORKING_BLOCKED_A);
   #ALARM_AUX := NOT ("M_ONE" AND NOT #ALARM_AUX AND NOT "DB16000_OPC_UA_TRIGGER_ALARM".CLIENT.U2_STA2_MEAS.ALARMS.PROFILER_CONFIG_A AND NOT "DB16000_OPC_UA_TRIGGER_ALARM".CLIENT.U2_STA2_MEAS.ALARMS.ANALYZER_CONFIG_A AND NOT "DB16000_OPC_UA_TRIGGER_ALARM".CLIENT.U2_STA2_MEAS.ALARMS.DMC_STRUCTURE_A AND NOT "DB16000_OPC_UA_TRIGGER_ALARM".CLIENT.U2_STA2_MEAS.ALARMS.ACQUISITION_A AND NOT "DB16000_OPC_UA_TRIGGER_ALARM".CLIENT.U2_STA2_MEAS.ALARMS.PROFILER_INIT_A AND NOT "DB16000_OPC_UA_TRIGGER_ALARM".CLIENT.U2_STA2_MEAS.ALARMS.UMBRELLA_A AND NOT "DB16000_OPC_UA_TRIGGER_ALARM".CLIENT.U2_STA2_MEAS.ALARMS.RUNOUT_A AND NOT "DB16000_OPC_UA_TRIGGER_ALARM".CLIENT.U2_STA2_MEAS.ALARMS.LAYER_GROWTH_A AND NOT "DB16000_OPC_UA_TRIGGER_ALARM".CLIENT.U2_STA2_MEAS.ALARMS.SURFACE_DEFECTS_A AND NOT "DB16000_OPC_UA_TRIGGER_ALARM".CLIENT.U2_STA2_MEAS.ALARMS.STORAGE_A AND NOT "DB16000_OPC_UA_TRIGGER_ALARM".CLIENT.U2_STA2_MEAS.ALARMS.CALIBRATION_MISSING_FIX_1_A AND NOT "DB16000_OPC_UA_TRIGGER_ALARM".CLIENT.U2_STA2_MEAS.ALARMS.CALIBRATION_MISSING_FIX_2_A AND NOT "DB16000_OPC_UA_TRIGGER_ALARM".CLIENT.U2_STA2_MEAS.ALARMS.CALIBRATION_MISSING_FIX_3_A AND NOT "DB16000_OPC_UA_TRIGGER_ALARM".CLIENT.U2_STA2_MEAS.ALARMS.CALIBRATION_MISSING_FIX_4_A AND NOT "DB16000_OPC_UA_TRIGGER_ALARM".CLIENT.U2_STA2_MEAS.ALARMS.CALIBRATION_PROC_A AND NOT "DB16000_OPC_UA_TRIGGER_ALARM".CLIENT.U2_STA2_MEAS.ALARMS.DATABASE_CONNECTION_A);
   #_w1 := NOT ("M_ONE" AND NOT #ALARM_AUX AND NOT "DB16000_OPC_UA_TRIGGER_ALARM".CLIENT.U2_STA2_MEAS.ALARMS.CALIBRATION_OUT_RANGE_FIX_1_A AND NOT "DB16000_OPC_UA_TRIGGER_ALARM".CLIENT.U2_STA2_MEAS.ALARMS.CALIBRATION_OUT_RANGE_FIX_2_A AND NOT "DB16000_OPC_UA_TRIGGER_ALARM".CLIENT.U2_STA2_MEAS.ALARMS.CALIBRATION_OUT_RANGE_FIX_3_A AND NOT "DB16000_OPC_UA_TRIGGER_ALARM".CLIENT.U2_STA2_MEAS.ALARMS.CALIBRATION_OUT_RANGE_FIX_4_A AND NOT "DB16000_OPC_UA_TRIGGER_ALARM".CLIENT.U2_STA2_MEAS.ALARMS.MEAS_INITIALIZING_SENSOR_A AND NOT "DB16000_OPC_UA_TRIGGER_ALARM".CLIENT.U2_STA2_MEAS.ALARMS.PLC_PC_MAJOR_VERSIONS_MISMATCH_A);
   IF #_w1 THEN "DB440_MACHINE_ALARM_DECODING".GLOBAL_ALARMS_MACHINE.ALARM_DECODING := 16013; END_IF;
   IF #_w1 AND "M_DUMMY_OFF" THEN
       "DB440_MACHINE_ALARM_DECODING".ALARMS_UNIT_2.ST2_MEASURING.IS_SEOC_ALARMS := TRUE;
   END_IF;
END_REGION

REGION Network 78: MAINTAIN POWDER ALARMS
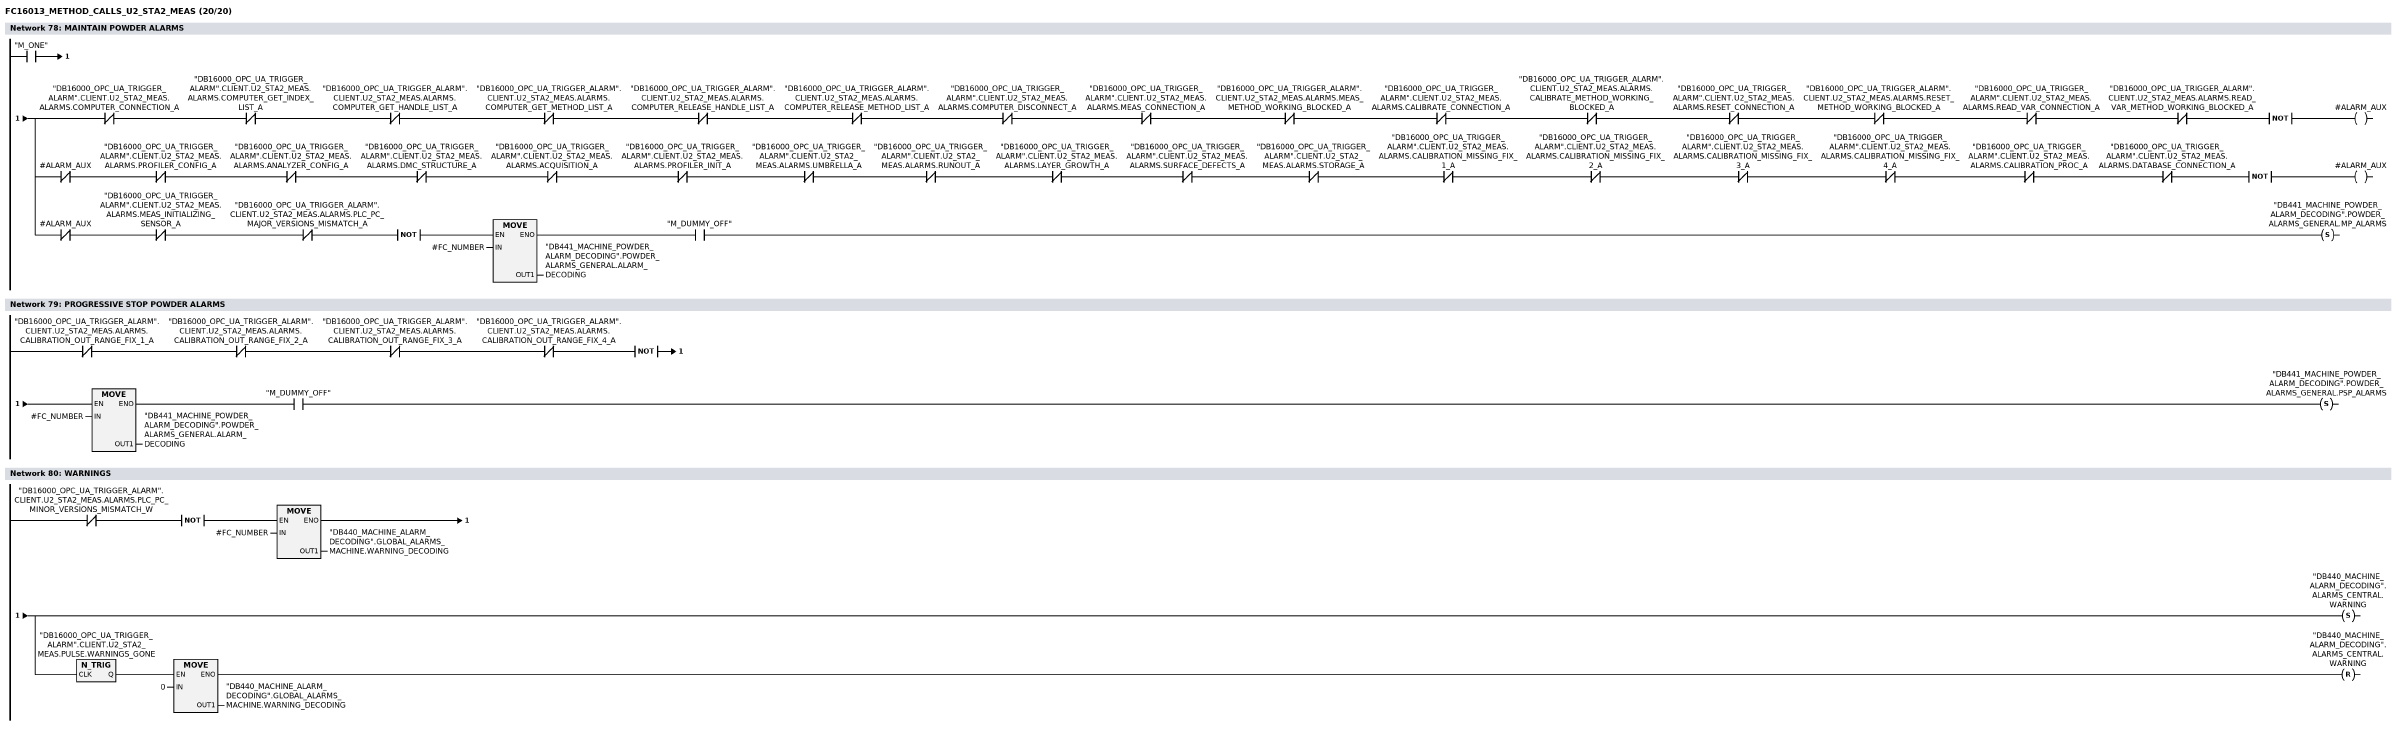
   RUNG wire#powerrail
      Contact( "M_ONE" )
      wire#w1
      I_Contact( "DB16000_OPC_UA_TRIGGER_ALARM".CLIENT.U2_STA2_MEAS.ALARMS.COMPUTER_CONNECTION_A )
      I_Contact( "DB16000_OPC_UA_TRIGGER_ALARM".CLIENT.U2_STA2_MEAS.ALARMS.COMPUTER_GET_INDEX_LIST_A )
      I_Contact( "DB16000_OPC_UA_TRIGGER_ALARM".CLIENT.U2_STA2_MEAS.ALARMS.COMPUTER_GET_HANDLE_LIST_A )
      I_Contact( "DB16000_OPC_UA_TRIGGER_ALARM".CLIENT.U2_STA2_MEAS.ALARMS.COMPUTER_GET_METHOD_LIST_A )
      I_Contact( "DB16000_OPC_UA_TRIGGER_ALARM".CLIENT.U2_STA2_MEAS.ALARMS.COMPUTER_RELEASE_HANDLE_LIST_A )
      I_Contact( "DB16000_OPC_UA_TRIGGER_ALARM".CLIENT.U2_STA2_MEAS.ALARMS.COMPUTER_RELEASE_METHOD_LIST_A )
      I_Contact( "DB16000_OPC_UA_TRIGGER_ALARM".CLIENT.U2_STA2_MEAS.ALARMS.COMPUTER_DISCONNECT_A )
      I_Contact( "DB16000_OPC_UA_TRIGGER_ALARM".CLIENT.U2_STA2_MEAS.ALARMS.MEAS_CONNECTION_A )
      I_Contact( "DB16000_OPC_UA_TRIGGER_ALARM".CLIENT.U2_STA2_MEAS.ALARMS.MEAS_METHOD_WORKING_BLOCKED_A )
      I_Contact( "DB16000_OPC_UA_TRIGGER_ALARM".CLIENT.U2_STA2_MEAS.ALARMS.CALIBRATE_CONNECTION_A )
      I_Contact( "DB16000_OPC_UA_TRIGGER_ALARM".CLIENT.U2_STA2_MEAS.ALARMS.CALIBRATE_METHOD_WORKING_BLOCKED_A )
      I_Contact( "DB16000_OPC_UA_TRIGGER_ALARM".CLIENT.U2_STA2_MEAS.ALARMS.RESET_CONNECTION_A )
      I_Contact( "DB16000_OPC_UA_TRIGGER_ALARM".CLIENT.U2_STA2_MEAS.ALARMS.RESET_METHOD_WORKING_BLOCKED_A )
      I_Contact( "DB16000_OPC_UA_TRIGGER_ALARM".CLIENT.U2_STA2_MEAS.ALARMS.READ_VAR_CONNECTION_A )
      I_Contact( "DB16000_OPC_UA_TRIGGER_ALARM".CLIENT.U2_STA2_MEAS.ALARMS.READ_VAR_METHOD_WORKING_BLOCKED_A )
      Not()
      Coil( #ALARM_AUX )
   END_RUNG
   RUNG wire#w1
      I_Contact( #ALARM_AUX )
      I_Contact( "DB16000_OPC_UA_TRIGGER_ALARM".CLIENT.U2_STA2_MEAS.ALARMS.PROFILER_CONFIG_A )
      I_Contact( "DB16000_OPC_UA_TRIGGER_ALARM".CLIENT.U2_STA2_MEAS.ALARMS.ANALYZER_CONFIG_A )
      I_Contact( "DB16000_OPC_UA_TRIGGER_ALARM".CLIENT.U2_STA2_MEAS.ALARMS.DMC_STRUCTURE_A )
      I_Contact( "DB16000_OPC_UA_TRIGGER_ALARM".CLIENT.U2_STA2_MEAS.ALARMS.ACQUISITION_A )
      I_Contact( "DB16000_OPC_UA_TRIGGER_ALARM".CLIENT.U2_STA2_MEAS.ALARMS.PROFILER_INIT_A )
      I_Contact( "DB16000_OPC_UA_TRIGGER_ALARM".CLIENT.U2_STA2_MEAS.ALARMS.UMBRELLA_A )
      I_Contact( "DB16000_OPC_UA_TRIGGER_ALARM".CLIENT.U2_STA2_MEAS.ALARMS.RUNOUT_A )
      I_Contact( "DB16000_OPC_UA_TRIGGER_ALARM".CLIENT.U2_STA2_MEAS.ALARMS.LAYER_GROWTH_A )
      I_Contact( "DB16000_OPC_UA_TRIGGER_ALARM".CLIENT.U2_STA2_MEAS.ALARMS.SURFACE_DEFECTS_A )
      I_Contact( "DB16000_OPC_UA_TRIGGER_ALARM".CLIENT.U2_STA2_MEAS.ALARMS.STORAGE_A )
      I_Contact( "DB16000_OPC_UA_TRIGGER_ALARM".CLIENT.U2_STA2_MEAS.ALARMS.CALIBRATION_MISSING_FIX_1_A )
      I_Contact( "DB16000_OPC_UA_TRIGGER_ALARM".CLIENT.U2_STA2_MEAS.ALARMS.CALIBRATION_MISSING_FIX_2_A )
      I_Contact( "DB16000_OPC_UA_TRIGGER_ALARM".CLIENT.U2_STA2_MEAS.ALARMS.CALIBRATION_MISSING_FIX_3_A )
      I_Contact( "DB16000_OPC_UA_TRIGGER_ALARM".CLIENT.U2_STA2_MEAS.ALARMS.CALIBRATION_MISSING_FIX_4_A )
      I_Contact( "DB16000_OPC_UA_TRIGGER_ALARM".CLIENT.U2_STA2_MEAS.ALARMS.CALIBRATION_PROC_A )
      I_Contact( "DB16000_OPC_UA_TRIGGER_ALARM".CLIENT.U2_STA2_MEAS.ALARMS.DATABASE_CONNECTION_A )
      Not()
      Coil( #ALARM_AUX )
   END_RUNG
   RUNG wire#w1
      I_Contact( #ALARM_AUX )
      I_Contact( "DB16000_OPC_UA_TRIGGER_ALARM".CLIENT.U2_STA2_MEAS.ALARMS.MEAS_INITIALIZING_SENSOR_A )
      I_Contact( "DB16000_OPC_UA_TRIGGER_ALARM".CLIENT.U2_STA2_MEAS.ALARMS.PLC_PC_MAJOR_VERSIONS_MISMATCH_A )
      Not()
      Move(in := #FC_NUMBER, out1 => "DB441_MACHINE_POWDER_ALARM_DECODING".POWDER_ALARMS_GENERAL.ALARM_DECODING)
      Contact( "M_DUMMY_OFF" )
      S_Coil( "DB441_MACHINE_POWDER_ALARM_DECODING".POWDER_ALARMS_GENERAL.MP_ALARMS )
   END_RUNG
   // the same network as SCL:
   #ALARM_AUX := NOT ("M_ONE" AND NOT "DB16000_OPC_UA_TRIGGER_ALARM".CLIENT.U2_STA2_MEAS.ALARMS.COMPUTER_CONNECTION_A AND NOT "DB16000_OPC_UA_TRIGGER_ALARM".CLIENT.U2_STA2_MEAS.ALARMS.COMPUTER_GET_INDEX_LIST_A AND NOT "DB16000_OPC_UA_TRIGGER_ALARM".CLIENT.U2_STA2_MEAS.ALARMS.COMPUTER_GET_HANDLE_LIST_A AND NOT "DB16000_OPC_UA_TRIGGER_ALARM".CLIENT.U2_STA2_MEAS.ALARMS.COMPUTER_GET_METHOD_LIST_A AND NOT "DB16000_OPC_UA_TRIGGER_ALARM".CLIENT.U2_STA2_MEAS.ALARMS.COMPUTER_RELEASE_HANDLE_LIST_A AND NOT "DB16000_OPC_UA_TRIGGER_ALARM".CLIENT.U2_STA2_MEAS.ALARMS.COMPUTER_RELEASE_METHOD_LIST_A AND NOT "DB16000_OPC_UA_TRIGGER_ALARM".CLIENT.U2_STA2_MEAS.ALARMS.COMPUTER_DISCONNECT_A AND NOT "DB16000_OPC_UA_TRIGGER_ALARM".CLIENT.U2_STA2_MEAS.ALARMS.MEAS_CONNECTION_A AND NOT "DB16000_OPC_UA_TRIGGER_ALARM".CLIENT.U2_STA2_MEAS.ALARMS.MEAS_METHOD_WORKING_BLOCKED_A AND NOT "DB16000_OPC_UA_TRIGGER_ALARM".CLIENT.U2_STA2_MEAS.ALARMS.CALIBRATE_CONNECTION_A AND NOT "DB16000_OPC_UA_TRIGGER_ALARM".CLIENT.U2_STA2_MEAS.ALARMS.CALIBRATE_METHOD_WORKING_BLOCKED_A AND NOT "DB16000_OPC_UA_TRIGGER_ALARM".CLIENT.U2_STA2_MEAS.ALARMS.RESET_CONNECTION_A AND NOT "DB16000_OPC_UA_TRIGGER_ALARM".CLIENT.U2_STA2_MEAS.ALARMS.RESET_METHOD_WORKING_BLOCKED_A AND NOT "DB16000_OPC_UA_TRIGGER_ALARM".CLIENT.U2_STA2_MEAS.ALARMS.READ_VAR_CONNECTION_A AND NOT "DB16000_OPC_UA_TRIGGER_ALARM".CLIENT.U2_STA2_MEAS.ALARMS.READ_VAR_METHOD_WORKING_BLOCKED_A);
   #ALARM_AUX := NOT ("M_ONE" AND NOT #ALARM_AUX AND NOT "DB16000_OPC_UA_TRIGGER_ALARM".CLIENT.U2_STA2_MEAS.ALARMS.PROFILER_CONFIG_A AND NOT "DB16000_OPC_UA_TRIGGER_ALARM".CLIENT.U2_STA2_MEAS.ALARMS.ANALYZER_CONFIG_A AND NOT "DB16000_OPC_UA_TRIGGER_ALARM".CLIENT.U2_STA2_MEAS.ALARMS.DMC_STRUCTURE_A AND NOT "DB16000_OPC_UA_TRIGGER_ALARM".CLIENT.U2_STA2_MEAS.ALARMS.ACQUISITION_A AND NOT "DB16000_OPC_UA_TRIGGER_ALARM".CLIENT.U2_STA2_MEAS.ALARMS.PROFILER_INIT_A AND NOT "DB16000_OPC_UA_TRIGGER_ALARM".CLIENT.U2_STA2_MEAS.ALARMS.UMBRELLA_A AND NOT "DB16000_OPC_UA_TRIGGER_ALARM".CLIENT.U2_STA2_MEAS.ALARMS.RUNOUT_A AND NOT "DB16000_OPC_UA_TRIGGER_ALARM".CLIENT.U2_STA2_MEAS.ALARMS.LAYER_GROWTH_A AND NOT "DB16000_OPC_UA_TRIGGER_ALARM".CLIENT.U2_STA2_MEAS.ALARMS.SURFACE_DEFECTS_A AND NOT "DB16000_OPC_UA_TRIGGER_ALARM".CLIENT.U2_STA2_MEAS.ALARMS.STORAGE_A AND NOT "DB16000_OPC_UA_TRIGGER_ALARM".CLIENT.U2_STA2_MEAS.ALARMS.CALIBRATION_MISSING_FIX_1_A AND NOT "DB16000_OPC_UA_TRIGGER_ALARM".CLIENT.U2_STA2_MEAS.ALARMS.CALIBRATION_MISSING_FIX_2_A AND NOT "DB16000_OPC_UA_TRIGGER_ALARM".CLIENT.U2_STA2_MEAS.ALARMS.CALIBRATION_MISSING_FIX_3_A AND NOT "DB16000_OPC_UA_TRIGGER_ALARM".CLIENT.U2_STA2_MEAS.ALARMS.CALIBRATION_MISSING_FIX_4_A AND NOT "DB16000_OPC_UA_TRIGGER_ALARM".CLIENT.U2_STA2_MEAS.ALARMS.CALIBRATION_PROC_A AND NOT "DB16000_OPC_UA_TRIGGER_ALARM".CLIENT.U2_STA2_MEAS.ALARMS.DATABASE_CONNECTION_A);
   #_w1 := NOT ("M_ONE" AND NOT #ALARM_AUX AND NOT "DB16000_OPC_UA_TRIGGER_ALARM".CLIENT.U2_STA2_MEAS.ALARMS.MEAS_INITIALIZING_SENSOR_A AND NOT "DB16000_OPC_UA_TRIGGER_ALARM".CLIENT.U2_STA2_MEAS.ALARMS.PLC_PC_MAJOR_VERSIONS_MISMATCH_A);
   IF #_w1 THEN
       "DB441_MACHINE_POWDER_ALARM_DECODING".POWDER_ALARMS_GENERAL.ALARM_DECODING := #FC_NUMBER;
   END_IF;
   IF #_w1 AND "M_DUMMY_OFF" THEN
       "DB441_MACHINE_POWDER_ALARM_DECODING".POWDER_ALARMS_GENERAL.MP_ALARMS := TRUE;
   END_IF;
END_REGION

REGION Network 79: PROGRESSIVE STOP POWDER ALARMS
   RUNG wire#powerrail
      I_Contact( "DB16000_OPC_UA_TRIGGER_ALARM".CLIENT.U2_STA2_MEAS.ALARMS.CALIBRATION_OUT_RANGE_FIX_1_A )
      I_Contact( "DB16000_OPC_UA_TRIGGER_ALARM".CLIENT.U2_STA2_MEAS.ALARMS.CALIBRATION_OUT_RANGE_FIX_2_A )
      I_Contact( "DB16000_OPC_UA_TRIGGER_ALARM".CLIENT.U2_STA2_MEAS.ALARMS.CALIBRATION_OUT_RANGE_FIX_3_A )
      I_Contact( "DB16000_OPC_UA_TRIGGER_ALARM".CLIENT.U2_STA2_MEAS.ALARMS.CALIBRATION_OUT_RANGE_FIX_4_A )
      Not()
      Move(in := #FC_NUMBER, out1 => "DB441_MACHINE_POWDER_ALARM_DECODING".POWDER_ALARMS_GENERAL.ALARM_DECODING)
      Contact( "M_DUMMY_OFF" )
      S_Coil( "DB441_MACHINE_POWDER_ALARM_DECODING".POWDER_ALARMS_GENERAL.PSP_ALARMS )
   END_RUNG
   // the same network as SCL:
   #_w1 := NOT (NOT "DB16000_OPC_UA_TRIGGER_ALARM".CLIENT.U2_STA2_MEAS.ALARMS.CALIBRATION_OUT_RANGE_FIX_1_A AND NOT "DB16000_OPC_UA_TRIGGER_ALARM".CLIENT.U2_STA2_MEAS.ALARMS.CALIBRATION_OUT_RANGE_FIX_2_A AND NOT "DB16000_OPC_UA_TRIGGER_ALARM".CLIENT.U2_STA2_MEAS.ALARMS.CALIBRATION_OUT_RANGE_FIX_3_A AND NOT "DB16000_OPC_UA_TRIGGER_ALARM".CLIENT.U2_STA2_MEAS.ALARMS.CALIBRATION_OUT_RANGE_FIX_4_A);
   IF #_w1 THEN
       "DB441_MACHINE_POWDER_ALARM_DECODING".POWDER_ALARMS_GENERAL.ALARM_DECODING := #FC_NUMBER;
   END_IF;
   IF #_w1 AND "M_DUMMY_OFF" THEN
       "DB441_MACHINE_POWDER_ALARM_DECODING".POWDER_ALARMS_GENERAL.PSP_ALARMS := TRUE;
   END_IF;
END_REGION

REGION Network 80: WARNINGS
   RUNG wire#powerrail
      I_Contact( "DB16000_OPC_UA_TRIGGER_ALARM".CLIENT.U2_STA2_MEAS.ALARMS.PLC_PC_MINOR_VERSIONS_MISMATCH_W )
      Not()
      Move(in := #FC_NUMBER, out1 => "DB440_MACHINE_ALARM_DECODING".GLOBAL_ALARMS_MACHINE.WARNING_DECODING)
      wire#w1
      S_Coil( "DB440_MACHINE_ALARM_DECODING".ALARMS_CENTRAL.WARNING )
   END_RUNG
   RUNG wire#w1
      N_Trig( "DB16000_OPC_UA_TRIGGER_ALARM".CLIENT.U2_STA2_MEAS.PULSE.WARNINGS_GONE )
      Move(in := 0, out1 => "DB440_MACHINE_ALARM_DECODING".GLOBAL_ALARMS_MACHINE.WARNING_DECODING)
      R_Coil( "DB440_MACHINE_ALARM_DECODING".ALARMS_CENTRAL.WARNING )
   END_RUNG
   // the same network as SCL:
   #_w1 := NOT (NOT "DB16000_OPC_UA_TRIGGER_ALARM".CLIENT.U2_STA2_MEAS.ALARMS.PLC_PC_MINOR_VERSIONS_MISMATCH_W);
   IF #_w1 THEN
       "DB440_MACHINE_ALARM_DECODING".GLOBAL_ALARMS_MACHINE.WARNING_DECODING := #FC_NUMBER;
       "DB440_MACHINE_ALARM_DECODING".ALARMS_CENTRAL.WARNING := TRUE;
   END_IF;
   #_w2 := NOT #_w1 AND "DB16000_OPC_UA_TRIGGER_ALARM".CLIENT.U2_STA2_MEAS.PULSE.WARNINGS_GONE;   // falling edge
   "DB16000_OPC_UA_TRIGGER_ALARM".CLIENT.U2_STA2_MEAS.PULSE.WARNINGS_GONE := #_w1;
   IF #_w2 THEN
       "DB440_MACHINE_ALARM_DECODING".GLOBAL_ALARMS_MACHINE.WARNING_DECODING := 0;
       "DB440_MACHINE_ALARM_DECODING".ALARMS_CENTRAL.WARNING := FALSE;
   END_IF;
END_REGION
END_FUNCTION
